// Check duration for each phase
positionExtrema := output.trajectory.profiles[0].positionExtrema();
AssertEquals_LREAL(0.04225334172441400082, positionExtrema.Tmax, 1E-9, message:='Profile[0] Tmax incorrect');
AssertEquals_LREAL(105.45722688838274905265, positionExtrema.Maximum, 1E-9, message:='Profile[0] maximum incorrect');
AssertEquals_LREAL(0.00000000000000000000, positionExtrema.Tmin, 1E-9, message:='Profile[0] Tmin incorrect');
AssertEquals_LREAL(92.10487433807648471884, positionExtrema.Minimum, 1E-9, message:='Profile[0] minimum incorrect');

positionExtrema := output.trajectory.profiles[1].positionExtrema();
AssertEquals_LREAL(0.00000000000000000000, positionExtrema.Tmax, 1E-9, message:='Profile[1] Tmax incorrect');
AssertEquals_LREAL(89.01461536061293600142, positionExtrema.Maximum, 1E-9, message:='Profile[1] maximum incorrect');
AssertEquals_LREAL(0.10861795461857774725, positionExtrema.Tmin, 1E-9, message:='Profile[1] Tmin incorrect');
AssertEquals_LREAL(56.54940187438580778689, positionExtrema.Minimum, 1E-9, message:='Profile[1] minimum incorrect');

positionExtrema := output.trajectory.profiles[2].positionExtrema();
AssertEquals_LREAL(0.00000000000000000000, positionExtrema.Tmax, 1E-9, message:='Profile[2] Tmax incorrect');
AssertEquals_LREAL(43.32328991111594973518, positionExtrema.Maximum, 1E-9, message:='Profile[2] maximum incorrect');
AssertEquals_LREAL(0.10861795461857774725, positionExtrema.Tmin, 1E-9, message:='Profile[2] Tmin incorrect');
AssertEquals_LREAL(5.30614662549113802470, positionExtrema.Minimum, 1E-9, message:='Profile[2] minimum incorrect');
   

TEST_FINISHED();
END_METHOD

METHOD Test_Trajectory_64
VAR_INST
  ruckig : Struckig.Ruckig(0.001);
  input : Struckig.InputParameter(3) := (
    Synchronization := SynchronizationType.TimeSync,        
    MaxVelocity := [ 2000.00000000000000000000, 2000.00000000000000000000, 2000.00000000000000000000 ],
    MaxAcceleration := [ 20000.00000000000000000000, 20000.00000000000000000000, 20000.00000000000000000000 ],
    MaxJerk := [ 800000.00000000000000000000, 800000.00000000000000000000, 800000.00000000000000000000 ],
    CurrentPosition := [ 84.12964321952199497900, 15.09477787023756434337, 10.23674324179428651860 ],
    CurrentVelocity := [ -970.87417203950269595225, -928.12491864862022339366, 286.06399288670468195050 ],
    CurrentAcceleration := [ 4961.60497362833666556980, 5135.12661885897978208959, 79.48669035600505594630 ],
    TargetPosition := [ -30.09864175377319384097, 39.92408869665283077666, 24.17762560090359613696 ],
    TargetVelocity := [ 0.00000000000000000000, 0.00000000000000000000, 0.00000000000000000000 ],
    TargetAcceleration := [ 0.00000000000000000000, 0.00000000000000000000, 0.00000000000000000000 ]
  );
  output : Struckig.OutputParameter;
  positionExtrema : Struckig.PositionExtremaDesc;
END_VAR
TEST('Trajectory_64');

ruckig.update(input, output);

// Check total duration of profiles
AssertEquals_LREAL(Expected := 0.17167999763375443867, Actual := output.Trajectory.Duration, DELTA := 1E-8, Message := 'Duration incorrect');

// Check duration for each phase
positionExtrema := output.trajectory.profiles[0].positionExtrema();
AssertEquals_LREAL(0.00000000000000000000, positionExtrema.Tmax, 1E-9, message:='Profile[0] Tmax incorrect');
AssertEquals_LREAL(84.12964321952199497900, positionExtrema.Maximum, 1E-9, message:='Profile[0] maximum incorrect');
AssertEquals_LREAL(0.17167999763375441091, positionExtrema.Tmin, 1E-9, message:='Profile[0] Tmin incorrect');
AssertEquals_LREAL(-30.09864175377319384097, positionExtrema.Minimum, 1E-9, message:='Profile[0] minimum incorrect');

positionExtrema := output.trajectory.profiles[1].positionExtrema();
AssertEquals_LREAL(0.17167999763375443867, positionExtrema.Tmax, 1E-9, message:='Profile[1] Tmax incorrect');
AssertEquals_LREAL(39.92408869665283077666, positionExtrema.Maximum, 1E-9, message:='Profile[1] maximum incorrect');
AssertEquals_LREAL(0.08124569148055139911, positionExtrema.Tmin, 1E-9, message:='Profile[1] Tmin incorrect');
AssertEquals_LREAL(-4.66763872582565753078, positionExtrema.Minimum, 1E-9, message:='Profile[1] minimum incorrect');

positionExtrema := output.trajectory.profiles[2].positionExtrema();
AssertEquals_LREAL(0.17167999763375443867, positionExtrema.Tmax, 1E-9, message:='Profile[2] Tmax incorrect');
AssertEquals_LREAL(24.17762560090359613696, positionExtrema.Maximum, 1E-9, message:='Profile[2] maximum incorrect');
AssertEquals_LREAL(0.00000000000000000000, positionExtrema.Tmin, 1E-9, message:='Profile[2] Tmin incorrect');
AssertEquals_LREAL(10.23674324179428651860, positionExtrema.Minimum, 1E-9, message:='Profile[2] minimum incorrect');
   

TEST_FINISHED();
END_METHOD

METHOD Test_Trajectory_65
VAR_INST
  ruckig : Struckig.Ruckig(0.001);
  input : Struckig.InputParameter(3) := (
    Synchronization := SynchronizationType.TimeSync,        
    MaxVelocity := [ 2000.00000000000000000000, 2000.00000000000000000000, 2000.00000000000000000000 ],
    MaxAcceleration := [ 20000.00000000000000000000, 20000.00000000000000000000, 20000.00000000000000000000 ],
    MaxJerk := [ 800000.00000000000000000000, 800000.00000000000000000000, 800000.00000000000000000000 ],
    CurrentPosition := [ 33.17628426446438538733, 50.00168428476928283999, 61.64263417164463021436 ],
    CurrentVelocity := [ -519.65995269471272877126, 66.93100559795539084007, -520.26416261644567384792 ],
    CurrentAcceleration := [ 3662.19439283437168342061, -8995.68879146701328863855, 4153.78894930269962060265 ],
    TargetPosition := [ 68.69261284366797326584, -66.97490772805458902894, -0.91414242050534255668 ],
    TargetVelocity := [ 0.00000000000000000000, 0.00000000000000000000, 0.00000000000000000000 ],
    TargetAcceleration := [ 0.00000000000000000000, 0.00000000000000000000, 0.00000000000000000000 ]
  );
  output : Struckig.OutputParameter;
  positionExtrema : Struckig.PositionExtremaDesc;
END_VAR
TEST('Trajectory_65');

ruckig.update(input, output);

// Check total duration of profiles
AssertEquals_LREAL(Expected := 0.17505526811503621665, Actual := output.Trajectory.Duration, DELTA := 1E-8, Message := 'Duration incorrect');

// Check duration for each phase
positionExtrema := output.trajectory.profiles[0].positionExtrema();
AssertEquals_LREAL(0.17505526811503624440, positionExtrema.Tmax, 1E-9, message:='Profile[0] Tmax incorrect');
AssertEquals_LREAL(68.69261284366797326584, positionExtrema.Maximum, 1E-9, message:='Profile[0] maximum incorrect');
AssertEquals_LREAL(0.04377678309027987352, positionExtrema.Tmin, 1E-9, message:='Profile[0] Tmin incorrect');
AssertEquals_LREAL(23.42380651880664998998, positionExtrema.Minimum, 1E-9, message:='Profile[0] minimum incorrect');

positionExtrema := output.trajectory.profiles[1].positionExtrema();
AssertEquals_LREAL(0.00589507367218594907, positionExtrema.Tmax, 1E-9, message:='Profile[1] Tmax incorrect');
AssertEquals_LREAL(50.21262355411419520124, positionExtrema.Maximum, 1E-9, message:='Profile[1] maximum incorrect');
AssertEquals_LREAL(0.17505526811503621665, positionExtrema.Tmin, 1E-9, message:='Profile[1] Tmin incorrect');
AssertEquals_LREAL(-66.97490772805458902894, positionExtrema.Minimum, 1E-9, message:='Profile[1] minimum incorrect');

positionExtrema := output.trajectory.profiles[2].positionExtrema();
AssertEquals_LREAL(0.00000000000000000000, positionExtrema.Tmax, 1E-9, message:='Profile[2] Tmax incorrect');
AssertEquals_LREAL(61.64263417164463021436, positionExtrema.Maximum, 1E-9, message:='Profile[2] maximum incorrect');
AssertEquals_LREAL(0.17505526750468464181, positionExtrema.Tmin, 1E-9, message:='Profile[2] Tmin incorrect');
AssertEquals_LREAL(-0.91414242050535987616, positionExtrema.Minimum, 1E-9, message:='Profile[2] minimum incorrect');
   

TEST_FINISHED();
END_METHOD

METHOD Test_Trajectory_HasTargetVelocity_HasTargetAcceleration_66
VAR_INST
  ruckig : Struckig.Ruckig(0.001);
  input : Struckig.InputParameter(3) := (
    Synchronization := SynchronizationType.TimeSync,        
    MaxVelocity := [ 2000.00000000000000000000, 2000.00000000000000000000, 2000.00000000000000000000 ],
    MaxAcceleration := [ 20000.00000000000000000000, 20000.00000000000000000000, 20000.00000000000000000000 ],
    MaxJerk := [ 800000.00000000000000000000, 800000.00000000000000000000, 800000.00000000000000000000 ],
    CurrentPosition := [ -48.80987185641822634352, 18.04364910313265113473, -24.74266082352920648191 ],
    CurrentVelocity := [ 988.42910759631240580347, -768.41448219800986407790, -207.75563249912386254437 ],
    CurrentAcceleration := [ 3735.71066306482680374756, -9295.98081225150599493645, 5866.28306601172880618833 ],
    TargetPosition := [ -12.17413972252995790768, 39.46835789725682275275, -82.53347662682273266910 ],
    TargetVelocity := [ 196.90336440418968777522, 718.33687283187941829965, -527.62167018153525077651 ],
    TargetAcceleration := [ -832.60782943610661277489, 502.29848616551748818893, 413.82241950646152872650 ]
  );
  output : Struckig.OutputParameter;
  positionExtrema : Struckig.PositionExtremaDesc;
END_VAR
TEST('Trajectory_HasTargetVelocity_HasTargetAcceleration_66');

ruckig.update(input, output);

// Check total duration of profiles
AssertEquals_LREAL(Expected := 0.15504630751390929833, Actual := output.Trajectory.Duration, DELTA := 1E-8, Message := 'Duration incorrect');

// Check duration for each phase
positionExtrema := output.trajectory.profiles[0].positionExtrema();
AssertEquals_LREAL(0.06757881268766546823, positionExtrema.Tmax, 1E-9, message:='Profile[0] Tmax incorrect');
AssertEquals_LREAL(-7.34951569385982939053, positionExtrema.Maximum, 1E-9, message:='Profile[0] maximum incorrect');
AssertEquals_LREAL(0.00000000000000000000, positionExtrema.Tmin, 1E-9, message:='Profile[0] Tmin incorrect');
AssertEquals_LREAL(-48.80987185641822634352, positionExtrema.Minimum, 1E-9, message:='Profile[0] minimum incorrect');

positionExtrema := output.trajectory.profiles[1].positionExtrema();
AssertEquals_LREAL(0.15504630751390929833, positionExtrema.Tmax, 1E-9, message:='Profile[1] Tmax incorrect');
AssertEquals_LREAL(39.46835789725682275275, positionExtrema.Maximum, 1E-9, message:='Profile[1] maximum incorrect');
AssertEquals_LREAL(0.03661997601531438024, positionExtrema.Tmin, 1E-9, message:='Profile[1] Tmin incorrect');
AssertEquals_LREAL(-9.78096891406795521107, positionExtrema.Minimum, 1E-9, message:='Profile[1] minimum incorrect');

positionExtrema := output.trajectory.profiles[2].positionExtrema();
AssertEquals_LREAL(0.00000000000000000000, positionExtrema.Tmax, 1E-9, message:='Profile[2] Tmax incorrect');
AssertEquals_LREAL(-24.74266082352920648191, positionExtrema.Maximum, 1E-9, message:='Profile[2] maximum incorrect');
AssertEquals_LREAL(0.15504630751390929833, positionExtrema.Tmin, 1E-9, message:='Profile[2] Tmin incorrect');
AssertEquals_LREAL(-82.53347662682273266910, positionExtrema.Minimum, 1E-9, message:='Profile[2] minimum incorrect');
   

TEST_FINISHED();
END_METHOD

METHOD Test_Trajectory_HasTargetAcceleration_67
VAR_INST
  ruckig : Struckig.Ruckig(0.001);
  input : Struckig.InputParameter(3) := (
    Synchronization := SynchronizationType.TimeSync,        
    MaxVelocity := [ 2000.00000000000000000000, 2000.00000000000000000000, 2000.00000000000000000000 ],
    MaxAcceleration := [ 20000.00000000000000000000, 20000.00000000000000000000, 20000.00000000000000000000 ],
    MaxJerk := [ 800000.00000000000000000000, 800000.00000000000000000000, 800000.00000000000000000000 ],
    CurrentPosition := [ -42.41545653101405832786, 92.92848487406354252016, 41.60376869401292765360 ],
    CurrentVelocity := [ 756.94781044141586789920, -102.29313054332476440322, -952.59491319783569451829 ],
    CurrentAcceleration := [ 2149.81876213580835610628, -9752.12830985097207303625, 1681.46952735132435918786 ],
    TargetPosition := [ 19.96620347711099441312, -33.22271553063156090957, 81.79650434185842300394 ],
    TargetVelocity := [ 0.00000000000000000000, 0.00000000000000000000, 0.00000000000000000000 ],
    TargetAcceleration := [ 338.30216212834284306155, -769.08223829335486243508, 288.55916186152558111644 ]
  );
  output : Struckig.OutputParameter;
  positionExtrema : Struckig.PositionExtremaDesc;
END_VAR
TEST('Trajectory_HasTargetAcceleration_67');

ruckig.update(input, output);

// Check total duration of profiles
AssertEquals_LREAL(Expected := 0.19427872815214472513, Actual := output.Trajectory.Duration, DELTA := 1E-8, Message := 'Duration incorrect');

// Check duration for each phase
positionExtrema := output.trajectory.profiles[0].positionExtrema();
AssertEquals_LREAL(0.19343297274682375031, positionExtrema.Tmax, 1E-9, message:='Profile[0] Tmax incorrect');
AssertEquals_LREAL(19.96624380849144131389, positionExtrema.Maximum, 1E-9, message:='Profile[0] maximum incorrect');
AssertEquals_LREAL(0.00000000000000000000, positionExtrema.Tmin, 1E-9, message:='Profile[0] Tmin incorrect');
AssertEquals_LREAL(-42.41545653101405832786, positionExtrema.Minimum, 1E-9, message:='Profile[0] minimum incorrect');

positionExtrema := output.trajectory.profiles[1].positionExtrema();
AssertEquals_LREAL(0.00000000000000000000, positionExtrema.Tmax, 1E-9, message:='Profile[1] Tmax incorrect');
AssertEquals_LREAL(92.92848487406354252016, positionExtrema.Maximum, 1E-9, message:='Profile[1] maximum incorrect');
AssertEquals_LREAL(0.19235602255641195968, positionExtrema.Tmin, 1E-9, message:='Profile[1] Tmin incorrect');
AssertEquals_LREAL(-33.22318938742549221388, positionExtrema.Minimum, 1E-9, message:='Profile[1] minimum incorrect');

positionExtrema := output.trajectory.profiles[2].positionExtrema();
AssertEquals_LREAL(0.19355733024749061100, positionExtrema.Tmax, 1E-9, message:='Profile[2] Tmax incorrect');
AssertEquals_LREAL(81.79652937027475445575, positionExtrema.Maximum, 1E-9, message:='Profile[2] maximum incorrect');
AssertEquals_LREAL(0.02289816309081084411, positionExtrema.Tmin, 1E-9, message:='Profile[2] Tmin incorrect');
AssertEquals_LREAL(21.83272724782310802993, positionExtrema.Minimum, 1E-9, message:='Profile[2] minimum incorrect');
   

TEST_FINISHED();
END_METHOD

METHOD Test_Trajectory_68
VAR_INST
  ruckig : Struckig.Ruckig(0.001);
  input : Struckig.InputParameter(3) := (
    Synchronization := SynchronizationType.TimeSync,        
    MaxVelocity := [ 2000.00000000000000000000, 2000.00000000000000000000, 2000.00000000000000000000 ],
    MaxAcceleration := [ 20000.00000000000000000000, 20000.00000000000000000000, 20000.00000000000000000000 ],
    MaxJerk := [ 800000.00000000000000000000, 800000.00000000000000000000, 800000.00000000000000000000 ],
    CurrentPosition := [ 40.62614323446814523777, 62.35469594204587906461, 24.25299098284108367807 ],
    CurrentVelocity := [ 953.39433299337724747602, 990.56715267728145590809, -738.17109364107295732538 ],
    CurrentAcceleration := [ 3444.24110064584601786919, 3257.77518810100627888460, 851.25313620111410273239 ],
    TargetPosition := [ -19.90968527499555307259, -93.17120052432892407523, -41.77005066216172934901 ],
    TargetVelocity := [ 0.00000000000000000000, 0.00000000000000000000, 0.00000000000000000000 ],
    TargetAcceleration := [ 0.00000000000000000000, 0.00000000000000000000, 0.00000000000000000000 ]
  );
  output : Struckig.OutputParameter;
  positionExtrema : Struckig.PositionExtremaDesc;
END_VAR
TEST('Trajectory_68');

ruckig.update(input, output);

// Check total duration of profiles
AssertEquals_LREAL(Expected := 0.27894619941724319023, Actual := output.Trajectory.Duration, DELTA := 1E-8, Message := 'Duration incorrect');

// Check duration for each phase
positionExtrema := output.trajectory.profiles[0].positionExtrema();
AssertEquals_LREAL(0.08122133382222911091, positionExtrema.Tmax, 1E-9, message:='Profile[0] Tmax incorrect');
AssertEquals_LREAL(76.63857184314483106391, positionExtrema.Maximum, 1E-9, message:='Profile[0] maximum incorrect');
AssertEquals_LREAL(0.27894619941724324574, positionExtrema.Tmin, 1E-9, message:='Profile[0] Tmin incorrect');
AssertEquals_LREAL(-19.90968527499555307259, positionExtrema.Minimum, 1E-9, message:='Profile[0] minimum incorrect');

positionExtrema := output.trajectory.profiles[1].positionExtrema();
AssertEquals_LREAL(0.02907221898512625524, positionExtrema.Tmax, 1E-9, message:='Profile[1] Tmax incorrect');
AssertEquals_LREAL(89.25318532542951288633, positionExtrema.Maximum, 1E-9, message:='Profile[1] maximum incorrect');
AssertEquals_LREAL(0.27894619941724319023, positionExtrema.Tmin, 1E-9, message:='Profile[1] Tmin incorrect');
AssertEquals_LREAL(-93.17120052432892407523, positionExtrema.Minimum, 1E-9, message:='Profile[1] minimum incorrect');

positionExtrema := output.trajectory.profiles[2].positionExtrema();
AssertEquals_LREAL(0.00000000000000000000, positionExtrema.Tmax, 1E-9, message:='Profile[2] Tmax incorrect');
AssertEquals_LREAL(24.25299098284108367807, positionExtrema.Maximum, 1E-9, message:='Profile[2] maximum incorrect');
AssertEquals_LREAL(0.27894619941724324574, positionExtrema.Tmin, 1E-9, message:='Profile[2] Tmin incorrect');
AssertEquals_LREAL(-41.77005066216172934901, positionExtrema.Minimum, 1E-9, message:='Profile[2] minimum incorrect');
   

TEST_FINISHED();
END_METHOD

METHOD Test_Trajectory_HasTargetVelocity_69
VAR_INST
  ruckig : Struckig.Ruckig(0.001);
  input : Struckig.InputParameter(3) := (
    Synchronization := SynchronizationType.TimeSync,        
    MaxVelocity := [ 2000.00000000000000000000, 2000.00000000000000000000, 2000.00000000000000000000 ],
    MaxAcceleration := [ 20000.00000000000000000000, 20000.00000000000000000000, 20000.00000000000000000000 ],
    MaxJerk := [ 800000.00000000000000000000, 800000.00000000000000000000, 800000.00000000000000000000 ],
    CurrentPosition := [ 57.27064181935406850243, 60.77262566521827125143, 62.27255646349433959585 ],
    CurrentVelocity := [ 537.97467176664963517396, -420.66138587481805188872, -215.06636530667026363517 ],
    CurrentAcceleration := [ -1444.96134368556158733554, -9785.35194497229167609476, -7380.59859225371474167332 ],
    TargetPosition := [ -63.84344825014372304395, -56.97669545923665168630, -22.85605311820776819332 ],
    TargetVelocity := [ -201.51935759086109101190, 630.98179272467473310826, 276.24214614430115943833 ],
    TargetAcceleration := [ 0.00000000000000000000, 0.00000000000000000000, 0.00000000000000000000 ]
  );
  output : Struckig.OutputParameter;
  positionExtrema : Struckig.PositionExtremaDesc;
END_VAR
TEST('Trajectory_HasTargetVelocity_69');

ruckig.update(input, output);

// Check total duration of profiles
AssertEquals_LREAL(Expected := 0.20486873141224784534, Actual := output.Trajectory.Duration, DELTA := 1E-8, Message := 'Duration incorrect');

// Check duration for each phase
positionExtrema := output.trajectory.profiles[0].positionExtrema();
AssertEquals_LREAL(0.02319379832039304701, positionExtrema.Tmax, 1E-9, message:='Profile[0] Tmax incorrect');
AssertEquals_LREAL(67.69603683932946580626, positionExtrema.Maximum, 1E-9, message:='Profile[0] maximum incorrect');
AssertEquals_LREAL(0.20486873141224784534, positionExtrema.Tmin, 1E-9, message:='Profile[0] Tmin incorrect');
AssertEquals_LREAL(-63.84344825014372304395, positionExtrema.Minimum, 1E-9, message:='Profile[0] minimum incorrect');

positionExtrema := output.trajectory.profiles[1].positionExtrema();
AssertEquals_LREAL(0.00000000000000000000, positionExtrema.Tmax, 1E-9, message:='Profile[1] Tmax incorrect');
AssertEquals_LREAL(60.77262566521827125143, positionExtrema.Maximum, 1E-9, message:='Profile[1] maximum incorrect');
AssertEquals_LREAL(0.17986873141224785089, positionExtrema.Tmin, 1E-9, message:='Profile[1] Tmin incorrect');
AssertEquals_LREAL(-70.66790694402018857545, positionExtrema.Minimum, 1E-9, message:='Profile[1] minimum incorrect');

positionExtrema := output.trajectory.profiles[2].positionExtrema();
AssertEquals_LREAL(0.00000000000000000000, positionExtrema.Tmax, 1E-9, message:='Profile[2] Tmax incorrect');
AssertEquals_LREAL(62.27255646349433959585, positionExtrema.Maximum, 1E-9, message:='Profile[2] maximum incorrect');
AssertEquals_LREAL(0.17986873141224782313, positionExtrema.Tmin, 1E-9, message:='Profile[2] Tmin incorrect');
AssertEquals_LREAL(-27.67877343848196147746, positionExtrema.Minimum, 1E-9, message:='Profile[2] minimum incorrect');
   

TEST_FINISHED();
END_METHOD

METHOD Test_Trajectory_HasTargetVelocity_HasTargetAcceleration_70
VAR_INST
  ruckig : Struckig.Ruckig(0.001);
  input : Struckig.InputParameter(3) := (
    Synchronization := SynchronizationType.TimeSync,        
    MaxVelocity := [ 2000.00000000000000000000, 2000.00000000000000000000, 2000.00000000000000000000 ],
    MaxAcceleration := [ 20000.00000000000000000000, 20000.00000000000000000000, 20000.00000000000000000000 ],
    MaxJerk := [ 800000.00000000000000000000, 800000.00000000000000000000, 800000.00000000000000000000 ],
    CurrentPosition := [ -92.33184858939047501281, 71.73781926022004995502, -55.27032026177170109804 ],
    CurrentVelocity := [ -952.87828015244156176777, -234.88833123485505893768, 123.27287252024666486250 ],
    CurrentAcceleration := [ -7266.87319497806674917229, -1917.48167665642540669069, -9579.01136324118306220043 ],
    TargetPosition := [ -64.62381428735777433303, 58.03768693667834099870, 63.08437907080863737974 ],
    TargetVelocity := [ 812.70256182329512739670, -863.39780178803880517080, -492.22548367060147711527 ],
    TargetAcceleration := [ 53.46404855095147468091, -729.77327604858464837889, -373.83030360848226791859 ]
  );
  output : Struckig.OutputParameter;
  positionExtrema : Struckig.PositionExtremaDesc;
END_VAR
TEST('Trajectory_HasTargetVelocity_HasTargetAcceleration_70');

ruckig.update(input, output);

// Check total duration of profiles
AssertEquals_LREAL(Expected := 0.22013991649512543169, Actual := output.Trajectory.Duration, DELTA := 1E-8, Message := 'Duration incorrect');

// Check duration for each phase
positionExtrema := output.trajectory.profiles[0].positionExtrema();
AssertEquals_LREAL(0.22013991649512543169, positionExtrema.Tmax, 1E-9, message:='Profile[0] Tmax incorrect');
AssertEquals_LREAL(-64.62381428735777433303, positionExtrema.Maximum, 1E-9, message:='Profile[0] maximum incorrect');
AssertEquals_LREAL(0.08266151031223724355, positionExtrema.Tmin, 1E-9, message:='Profile[0] Tmin incorrect');
AssertEquals_LREAL(-135.90053229571682891219, positionExtrema.Minimum, 1E-9, message:='Profile[0] minimum incorrect');

positionExtrema := output.trajectory.profiles[1].positionExtrema();
AssertEquals_LREAL(0.16474949862477941687, positionExtrema.Tmax, 1E-9, message:='Profile[1] Tmax incorrect');
AssertEquals_LREAL(86.19544571063090643293, positionExtrema.Maximum, 1E-9, message:='Profile[1] maximum incorrect');
AssertEquals_LREAL(0.22013991649512543169, positionExtrema.Tmin, 1E-9, message:='Profile[1] Tmin incorrect');
AssertEquals_LREAL(58.03768693667834099870, positionExtrema.Minimum, 1E-9, message:='Profile[1] minimum incorrect');

positionExtrema := output.trajectory.profiles[2].positionExtrema();
AssertEquals_LREAL(0.19560720437463602339, positionExtrema.Tmax, 1E-9, message:='Profile[2] Tmax incorrect');
AssertEquals_LREAL(73.07882819675037922025, positionExtrema.Maximum, 1E-9, message:='Profile[2] maximum incorrect');
AssertEquals_LREAL(0.00000000000000000000, positionExtrema.Tmin, 1E-9, message:='Profile[2] Tmin incorrect');
AssertEquals_LREAL(-55.27032026177170109804, positionExtrema.Minimum, 1E-9, message:='Profile[2] minimum incorrect');
   

TEST_FINISHED();
END_METHOD

END_FUNCTION_BLOCK

(* stored: Version 1.1.0.1, ProductVersion 3.1.4024.9
   POU GeneratedTest: Id {8a002d40-1b8b-4a36-917f-04dd149a7db3}, SpecialFunc None
   Method Test_Trajectory_HasTargetAcceleration_1: Id {cb021cd2-1eb2-497e-92b0-13ba4b162b4d}
   Method Test_Trajectory_2: Id {feb7deb7-240d-4725-bc69-7e49533aac11}
   Method Test_Trajectory_HasTargetVelocity_3: Id {156e9032-b854-4120-85a4-c009510a36d1}
   Method Test_Trajectory_HasTargetVelocity_4: Id {26e930ca-eaec-46e3-a2b8-44e478f3b43a}
   Method Test_Trajectory_5: Id {13f76fd9-ef01-482e-9806-d541fd789409}
   Method Test_Trajectory_6: Id {e4769e83-a70a-495b-8650-48473eb66061}
   Method Test_Trajectory_7: Id {f443cdcd-0a4e-4a5f-83c7-aa270d8c4f29}
   Method Test_Trajectory_HasTargetAcceleration_8: Id {3b045538-5e0c-4eba-ae88-0fe0e39c02f8}
   Method Test_Trajectory_HasTargetVelocity_9: Id {bd04899e-e39d-49c0-b3f2-1ff83c02e385}
   Method Test_Trajectory_HasTargetVelocity_HasTargetAcceleration_10: Id {1de954f0-0a2b-47c4-922d-2b812dcb585b}
   Method Test_Trajectory_HasTargetVelocity_HasTargetAcceleration_11: Id {13931c03-21c3-445e-8415-7b7006270f3c}
   Method Test_Trajectory_12: Id {58f9f3ea-5aa9-42a6-982d-d62f562beb42}
   Method Test_Trajectory_HasTargetVelocity_HasTargetAcceleration_13: Id {f57cc478-3ee7-4ec1-b0c5-b72080353083}
   Method Test_Trajectory_HasTargetVelocity_14: Id {df9c4481-6c05-4858-9785-c91265efb52b}
   Method Test_Trajectory_HasTargetVelocity_15: Id {2cecfef8-d2e2-495e-bebb-bc5a74fc5143}
   Method Test_Trajectory_16: Id {86edb4f5-1bc8-4378-bcbe-49b36e551e58}
   Method Test_Trajectory_HasTargetVelocity_17: Id {fddf6355-7ab1-4f8f-94fa-f02648228ffd}
   Method Test_Trajectory_HasTargetAcceleration_18: Id {87bf6721-83d8-4b32-966c-99ac4a78d639}
   Method Test_Trajectory_HasTargetVelocity_19: Id {12ac8376-83bf-4d7c-a523-0488d72cc5f9}
   Method Test_Trajectory_HasTargetVelocity_20: Id {39cf6ad3-ef5c-48de-9c5b-1a87835b971f}
   Method Test_Trajectory_HasTargetVelocity_21: Id {e41ac4cf-8c86-4d4a-9d1f-d9e5dba955a9}
   Method Test_Trajectory_HasTargetVelocity_22: Id {0921bf0c-1724-4feb-b2ce-f8a6875619ac}
   Method Test_Trajectory_HasTargetVelocity_HasTargetAcceleration_23: Id {3d231d1e-c57a-4510-b4e7-6f33a49c2702}
   Method Test_Trajectory_HasTargetVelocity_HasTargetAcceleration_24: Id {c2c01e64-dc44-49a9-bee8-b55016f0f163}
   Method Test_Trajectory_HasTargetVelocity_HasTargetAcceleration_25: Id {c7e311d2-5dfb-4e51-a566-218e5a52fa90}
   Method Test_Trajectory_HasTargetAcceleration_26: Id {78b2dd22-53cc-4816-80c8-7473b9a3d28e}
   Method Test_Trajectory_HasTargetVelocity_27: Id {5df7da38-6b62-4d63-9965-5d59c1422b2d}
   Method Test_Trajectory_HasTargetVelocity_HasTargetAcceleration_28: Id {8e96e48c-6489-4b32-8734-dd18b59c5214}
   Method Test_Trajectory_HasTargetAcceleration_29: Id {8b14fd82-1380-457d-b2f1-c9b66dfd3987}
   Method Test_Trajectory_30: Id {4de81f97-6bfa-40ca-a367-0928a45b7b8c}
   Method Test_Trajectory_HasTargetVelocity_HasTargetAcceleration_31: Id {6ea2f4dd-29ae-4d36-8696-0b13eb748d83}
   Method Test_Trajectory_32: Id {80fcbbf3-69f2-46af-adc1-894cfdbbce94}
   Method Test_Trajectory_33: Id {700ca3c0-7a65-472c-a638-df977d35440e}
   Method Test_Trajectory_HasTargetVelocity_34: Id {6e6b4c5e-4c0b-4ee4-bf64-d2e11c192029}
   Method Test_Trajectory_HasTargetVelocity_35: Id {d63d6fa5-15d2-4e6c-a421-4881ea92e8f9}
   Method Test_Trajectory_HasTargetVelocity_36: Id {a29cd5cf-ffe9-4f03-a489-be3bc1df9990}
   Method Test_Trajectory_HasTargetAcceleration_37: Id {aaa4a0ba-5130-46a0-8ffa-b27e907e8bd6}
   Method Test_Trajectory_HasTargetVelocity_HasTargetAcceleration_38: Id {ecebe997-7b6c-416e-84b7-df34f73be55b}
   Method Test_Trajectory_HasTargetAcceleration_39: Id {e83eeeda-2b9f-4161-acea-d8df35bcdc43}
   Method Test_Trajectory_40: Id {0583eeff-b654-4173-ae02-db44e8cebcd8}
   Method Test_Trajectory_HasTargetVelocity_HasTargetAcceleration_41: Id {21990934-9f5e-4c0c-955d-b5c7e30c5513}
   Method Test_Trajectory_HasTargetAcceleration_42: Id {50384466-d3d3-4855-9ae2-90b2a541f15f}
   Method Test_Trajectory_HasTargetAcceleration_43: Id {9f4afb81-5dec-45e2-b726-8c31dd42c704}
   Method Test_Trajectory_HasTargetVelocity_44: Id {56c96b0b-fe80-4943-91c9-1fdcb81a6624}
   Method Test_Trajectory_HasTargetVelocity_45: Id {ac33e000-d88d-4dfc-8992-a3f1cde5b407}
   Method Test_Trajectory_HasTargetVelocity_HasTargetAcceleration_46: Id {e687be06-98c9-46be-a957-a0e3424f8f2b}
   Method Test_Trajectory_HasTargetVelocity_HasTargetAcceleration_47: Id {4ab42851-4a77-4ce0-bb00-2db1043bcf55}
   Method Test_Trajectory_HasTargetVelocity_HasTargetAcceleration_48: Id {0dfcaf5e-82ec-4b4f-834b-a4f2a0637f24}
   Method Test_Trajectory_49: Id {72a5070e-83e4-4ffa-89e6-c521b0557d81}
   Method Test_Trajectory_HasTargetAcceleration_50: Id {83986aec-d8d3-44b7-9035-1a2fe458a6b4}
   Method Test_Trajectory_HasTargetVelocity_HasTargetAcceleration_51: Id {4910e5a2-2dd1-4c8d-a2ef-8b89e8d667fe}
   Method Test_Trajectory_HasTargetVelocity_HasTargetAcceleration_52: Id {053c2965-a6b9-4e9b-ad46-340e7ff2135e}
   Method Test_Trajectory_53: Id {faa24a53-3c24-444f-a082-779aa468a44d}
   Method Test_Trajectory_HasTargetVelocity_54: Id {dfe940ba-a224-4684-aa6d-862aaca9f029}
   Method Test_Trajectory_HasTargetVelocity_55: Id {0fbece0f-b41b-4f95-82e9-544a7b7e2adb}
   Method Test_Trajectory_HasTargetVelocity_HasTargetAcceleration_56: Id {6ece3637-3eaa-4618-b255-cacd99d912ee}
   Method Test_Trajectory_HasTargetAcceleration_57: Id {ebd797d2-0238-4938-8213-925fec703cb4}
   Method Test_Trajectory_HasTargetAcceleration_58: Id {8c3b9170-2f82-40b2-a80f-6e21d7c72dfc}
   Method Test_Trajectory_59: Id {a7494a40-e9ee-4ed7-b86c-d5f7b1b24137}
   Method Test_Trajectory_HasTargetVelocity_HasTargetAcceleration_60: Id {589d4460-1fb2-4240-a9c3-49da90ff47a6}
   Method Test_Trajectory_HasTargetVelocity_HasTargetAcceleration_61: Id {5f1a6e08-4af6-469c-94d5-ec075bc8a4a8}
   Method Test_Trajectory_62: Id {65ab1bc3-7c0d-4d67-930f-12ee3f027e42}
   Method Test_Trajectory_HasTargetAcceleration_63: Id {7118233b-6700-4746-a588-47b64f552e26}
   Method Test_Trajectory_64: Id {6c69e6af-4862-4376-b2e6-a16c5b250733}
   Method Test_Trajectory_65: Id {6e0e0934-027d-4357-8b2d-1ec83f92d0c2}
   Method Test_Trajectory_HasTargetVelocity_HasTargetAcceleration_66: Id {df551abb-ef94-48f0-bd6c-eb2644b2e42f}
   Method Test_Trajectory_HasTargetAcceleration_67: Id {f0f13fcd-666a-41d3-a599-05259ea711bc}
   Method Test_Trajectory_68: Id {893b900a-8ff0-42b8-a82e-528dfc832c4e}
   Method Test_Trajectory_HasTargetVelocity_69: Id {406457be-60fd-4e49-b447-3b03452fbb61}
   Method Test_Trajectory_HasTargetVelocity_HasTargetAcceleration_70: Id {2807c9fd-c227-412f-8b2d-45de94481f19} *)
